(* PLC project Guard Clauses Example.project, CODESYS CODESYS V3.5 SP20 Patch 1 *)
(* stored: creationDateTime 2025-06-03T09:33:49.8273024, modificationDateTime 2025-06-03T09:33:32.9902694 *)

PROGRAM Main
  VAR
    ConditionA : BOOL;
    ConditionB : BOOL;
    ConditionC : BOOL;
  END_VAR

                    
// Instead of this -->
IF ConditionA THEN
    IF ConditionB THEN
        IF NOT ConditionC THEN
            DoSomething();
        END_IF
    END_IF
END_IF


//----------------------------------------------------------------------------+

// Try this -->
IF NOT ConditionA THEN RETURN; END_IF
IF NOT ConditionB THEN RETURN; END_IF
IF ConditionC THEN RETURN; END_IF

DoSomething();




                  

METHOD DoSomething : BOOL
                          
                        
END_METHOD
END_PROGRAM

CONFIGURATION Device
  RESOURCE Application ON PLC
    TASK MainTask(INTERVAL := T#20ms, PRIORITY := 1);
    PROGRAM Main WITH MainTask : Main;
  END_RESOURCE
END_CONFIGURATION
